FUNCTION_BLOCK VVI_Pacemaker
  (* Standard: 61499-2 *)
  (* Version 0.1, 2014-00-19, Administrator, NE734EFZE6G0NVX *)
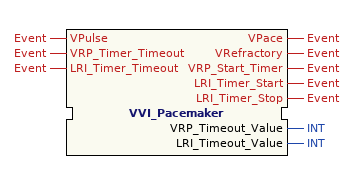
  EVENT_INPUT
    VPulse;
    VRP_Timer_Timeout;
    LRI_Timer_Timeout;
  END_EVENT
  EVENT_OUTPUT
    VPace;
    VRefractory;
    VRP_Start_Timer;
    LRI_Timer_Start;
    LRI_Timer_Stop;
  END_EVENT
  VAR_OUTPUT
    VRP_Timeout_Value : INT;
    LRI_Timeout_Value : INT;
  END_VAR
  FBS
    VVI_LRI : VVI_LRI;
    VVI_VRP : VVI_VRP;
  END_FBS
  EVENT_CONNECTIONS
    VPulse TO VVI_VRP.VPulse;
    VRP_Timer_Timeout TO VVI_VRP.VRP_Timer_Timeout;
    LRI_Timer_Timeout TO VVI_LRI.LRI_Timer_Timeout;
    VVI_LRI.VPace TO VPace;
    VVI_VRP.VRefractory TO VRefractory;
    VVI_VRP.VRP_Start_Timer TO VRP_Start_Timer;
    VVI_LRI.LRI_Timer_Start TO LRI_Timer_Start;
    VVI_LRI.LRI_Timer_Stop TO LRI_Timer_Stop;
    VVI_LRI.VPace TO VVI_VRP.VPace;
    VVI_VRP.VSense TO VVI_LRI.VSense;
  END_CONNECTIONS
  DATA_CONNECTIONS
    VVI_VRP.VRP_Timeout_Value TO VRP_Timeout_Value;
    VVI_LRI.LRI_Timeout_Value TO LRI_Timeout_Value;
  END_CONNECTIONS
END_FUNCTION_BLOCK
